FUNCTION proj2_TupleStruct_2: REAL
{ S7_Optimized_Access := 'false' }
    VAR_INPUT
        tuple: TupleStruct_2;
    END_VAR

BEGIN
    proj2_TupleStruct_2 := tuple.field2;
END_FUNCTION
